(* Generic data type used for Programs/Functions/Function Blocks to handle data in a generic way. *)
{attribute 'enable_dynamic_creation'}
TYPE ST_GENERIC EXTENDS __SYSTEM.AnyType :
STRUCT
	sValue : T_MaxString; 	// Data of parameter as a string for easy convertion.
END_STRUCT
END_TYPE

(* stored: Version 1.1.0.1, ProductVersion 3.1.4024.4
   DUT ST_GENERIC: Id {4f59ef17-3af4-404f-a2c8-af1971ec3536} *)
